(* PLC project  *)

CONFIGURATION Application
  RESOURCE Application ON PLC
    TASK SoftMotionPlanningTask(PRIORITY := 30);
    PROGRAM NCInterpreter WITH SoftMotionPlanningTask : NCInterpreter;
  END_RESOURCE
END_CONFIGURATION
